INTERFACE I_Sensor

PROPERTY IsActive : BOOL
GET
END_GET
END_PROPERTY

END_INTERFACE

(* stored: Version 1.1.0.1, ProductVersion 3.1.4024.9
   Itf I_Sensor: Id {bb361880-8c99-4cfa-9990-d76f12082fd8}
   Property IsActive: Id {39a95599-08fd-4822-83cd-db717370f9b7}
   Get Get: Id {b52d6804-b05f-4cd4-9561-96f176366373} *)
